// TwinCAT 3 PLC project Testing
// ProgramVersion: 3.1.4026.13
// libraries:
//   Tc2_Standard, * (Beckhoff Automation GmbH)
//   Tc2_System, * (Beckhoff Automation GmbH)
//   Tc3_Component, * (Zerlauth)
//   Tc3_Module, * (Beckhoff Automation GmbH)
//   Tc3_UnitTest, * (Zerlauth)
// project tree:
//   / PlcTask.TcTTO
//   POUs/ MAIN.TcPOU
//   Tests/ FB_ListComponentTests.TcPOU, FB_ListObjectTests.TcPOU, FB_ListStringTests.TcPOU (not stored), FB_MembersTests.TcPOU, FB_ComponentTests.TcPOU (not stored)
// (motion and I/O tree: see PLC project development)
// real-time tasks:
//   TASK PlcTask: cycle T#500ms, priority 21, ADS port 351
//   TASK UnitTestTask: cycle T#1ms, priority 1, ADS port 350
// variable links:

CONFIGURATION Testing
    RESOURCE PLC ON TwinCAT3
        TASK PlcTask(INTERVAL := T#1ms, PRIORITY := 1);
        PROGRAM MAIN WITH PlcTask : MAIN;
    END_RESOURCE
END_CONFIGURATION

// ---- POUs/MAIN.TcPOU
PROGRAM MAIN
VAR
	bInitialise: 			BOOL:= TRUE;
	bExecute: 				BOOL;
	fbTestsuites:			FB_Testsuites;
	fbListObject:			FB_ListObjectTests;
	fbListComponent:		FB_ListComponentTests;
	fbListString:			FB_ListStringTests;
	fbMembers:				FB_MembersTests;
	fbComponentTests:		FB_ComponentTests;
END_VAR

IF bInitialise THEN
	bInitialise:= FALSE;
	fbTestsuites.M_Add(fbListObject.fbTestsuite);
	fbTestsuites.M_Add(fbListComponent.fbTestsuite);
	fbTestsuites.M_Add(fbListString.fbTestsuite);
	fbTestsuites.M_Add(fbMembers.fbTestsuite);
	fbTestsuites.M_Add(fbComponentTests.fbTestsuite);
	fbTestsuites.P_Options.sFilePathName:= 'C:\report.xml';
END_IF

IF bExecute THEN
	bExecute:= fbTestsuites.M_Request(E_Base.Execute);
END_IF

fbTestsuites();


fbListObject();
fbListComponent();
fbListString();
fbMembers();
fbComponentTests();

END_PROGRAM

// ---- Tests/FB_ListObjectTests.TcPOU
FUNCTION_BLOCK FB_ListObjectTests EXTENDS 
VAR_INPUT
END_VAR
VAR_OUTPUT
	fbTestsuite:			FB_Testsuite;
END_VAR
VAR
	fbList:					Tc3_Component.FB_ListObject;
	fbObject:				Tc3_Component.FB_Component;
	iObject:				Tc3_Component.I_Object:= fbObject;
END_VAR

fbTestsuite.P_Property.M_Add('object', 'FB_ListObject');
fbTestsuite.P_Property.M_Add('name', 'Peter Zerlauth');

fbTestsuite();

CASE fbTestsuite.P_Testcase OF
	
	E_Testcase.Start:
		fbTestsuite.P_Assert.M_Equals_DINT(fbList.P_Length, 0, 'P_Length');
		fbTestsuite.M_Testcase('FB_ListObject', T#2S, 'fbList.P_Length', '', 10);	
		
	10:
		fbTestsuite.P_Assert.M_Equals_BOOL(fbList.M_Add(fbObject), TRUE, 'M_Add(fbObject)');
		fbTestsuite.M_Testcase('FB_ListObject', T#2S, 'fbList.M_Add(fbObject)', '', 20);
		
	20:
		fbTestsuite.P_Assert.M_Equals_DINT(fbList.P_Length, 1, 'P_Length');
		fbTestsuite.M_Testcase('FB_ListObject', T#2S, 'fbList.P_Length', '', 30);		
		
	30:
		fbTestsuite.P_Assert.M_Equals_DINT(fbList.M_Find(fbObject), 0, 'M_Find');
		fbTestsuite.M_Testcase('FB_ListObject', T#2S, 'fbList.M_Find(fbObject)', '', 40);
		
	40:

		fbTestsuite.P_Assert.M_Equals_BOOL(TRUE, __QUERYINTERFACE(fbList.M_Index(0), iObject), 'M_Index');
		fbTestsuite.M_Testcase('FB_ListObject', T#2S, 'fbList.M_Index(1)', '', 50);
		
	50:
		fbTestsuite.P_Assert.M_Equals_BOOL(fbList.M_Remove(fbObject), TRUE, 'M_Remove');
		fbTestsuite.M_Testcase('FB_ListObject', T#2S, 'fbList.M_Remove(fbObject', '', 60);		

	60:
		fbTestsuite.P_Assert.M_Equals_DINT(fbList.P_Length, 0, 'P_Length');
		fbTestsuite.M_Testcase('FB_ListObject', T#2S, 'fbList.P_Length', '', 70);
		
	70:
		fbTestsuite.P_Assert.M_Equals_BOOL(fbList.M_Add(fbObject), TRUE, 'M_Add(fbObject)');
		fbTestsuite.M_Testcase('FB_ListObject', T#2S, 'fbList.M_Add(fbObject)', '', 80);

	80:
		fbTestsuite.P_Assert.M_Equals_DINT(fbList.P_Length, 1, 'P_Length');
		fbTestsuite.M_Testcase('FB_ListObject', T#2S, 'fbList.P_Length', '', 90);
		
	90:
		fbTestsuite.P_Assert.M_Equals_BOOL(fbList.M_Clear(), TRUE, 'M_Clear()');
		fbTestsuite.M_Testcase('FB_ListObject', T#2S, 'fbList.M_Clear()', '', 100);		
	
	100:
		fbTestsuite.P_Assert.M_Equals_DINT(fbList.P_Length, 0, 'P_Length');
		fbTestsuite.M_Testcase('FB_ListObject', T#2S, 'fbList.P_Length', '', E_Testcase.Done);
		
	E_Testcase.Done:
		;
END_CASE

END_FUNCTION_BLOCK

// ---- Tests/FB_ListComponentTests.TcPOU
FUNCTION_BLOCK FB_ListComponentTests EXTENDS 
VAR_INPUT
END_VAR
VAR_OUTPUT
	fbTestsuite:			FB_Testsuite;
END_VAR
VAR
	fbList:					Tc3_Component.FB_ListComponent;
	fbObject:				Tc3_Component.FB_Component;
	iObject:				Tc3_Component.I_Element:= fbObject;
END_VAR

fbTestsuite.P_Property.M_Add('object', 'FB_ListComponent');
fbTestsuite.P_Property.M_Add('name', 'Peter Zerlauth');

fbTestsuite();

CASE fbTestsuite.P_Testcase OF
	
	E_Testcase.Start:
		fbTestsuite.P_Assert.M_Equals_DINT(fbList.P_Length, 0, 'P_Length');
		fbTestsuite.M_Testcase('FB_ListComponent', T#2S, 'fbList.P_Length', '', 10);	
		
	10:
		fbTestsuite.P_Assert.M_Equals_BOOL(fbList.M_Add(fbObject), TRUE, 'M_Add(fbObject)');
		fbTestsuite.M_Testcase('FB_ListComponent', T#2S, 'fbList.M_Add(fbObject)', '', 20);
		
	20:
		fbTestsuite.P_Assert.M_Equals_DINT(fbList.P_Length, 1, 'P_Length');
		fbTestsuite.M_Testcase('FB_ListComponent', T#2S, 'fbList.P_Length', '', 30);		
		
	30:
		fbTestsuite.P_Assert.M_Equals_DINT(fbList.M_Find(fbObject), 0, 'M_Find');
		fbTestsuite.M_Testcase('FB_ListComponent', T#2S, 'fbList.M_Find(fbObject)', '', 40);
		
	40:

		fbTestsuite.P_Assert.M_Equals_BOOL(TRUE, __QUERYINTERFACE(fbList.M_Index(0), iObject), 'M_Index');
		fbTestsuite.M_Testcase('FB_ListComponent', T#2S, 'fbList.M_Index(1)', '', 50);
		
	50:
		fbTestsuite.P_Assert.M_Equals_BOOL(fbList.M_Remove(fbObject), TRUE, 'M_Remove');
		fbTestsuite.M_Testcase('FB_ListComponent', T#2S, 'fbList.M_Remove(fbObject', '', 60);		

	60:
		fbTestsuite.P_Assert.M_Equals_DINT(fbList.P_Length, 0, 'P_Length');
		fbTestsuite.M_Testcase('FB_ListComponent', T#2S, 'fbList.P_Length', '', 70);
		
	70:
		fbTestsuite.P_Assert.M_Equals_BOOL(fbList.M_Add(fbObject), TRUE, 'M_Add(fbObject)');
		fbTestsuite.M_Testcase('FB_ListComponent', T#2S, 'fbList.M_Add(fbObject)', '', 80);

	80:
		fbTestsuite.P_Assert.M_Equals_DINT(fbList.P_Length, 1, 'P_Length');
		fbTestsuite.M_Testcase('FB_ListComponent', T#2S, 'fbList.P_Length', '', 90);
		
	90:
		fbTestsuite.P_Assert.M_Equals_BOOL(fbList.M_Clear(), TRUE, 'M_Clear()');
		fbTestsuite.M_Testcase('FB_ListComponent', T#2S, 'fbList.M_Clear()', '', 100);		
	
	100:
		fbTestsuite.P_Assert.M_Equals_DINT(fbList.P_Length, 0, 'P_Length');
		fbTestsuite.M_Testcase('FB_ListComponent', T#2S, 'fbList.P_Length', '', E_Testcase.Done);
		
	E_Testcase.Done:
		;
END_CASE

END_FUNCTION_BLOCK

// ---- Tests/FB_MembersTests.TcPOU
FUNCTION_BLOCK FB_MembersTests EXTENDS 
VAR_INPUT
END_VAR
VAR_OUTPUT
	fbTestsuite:			FB_Testsuite;
END_VAR
VAR
	fbList:					Tc3_Component.FB_Members;
	fbObject1:				Tc3_Component.FB_Component;
	fbObject2:				Tc3_Component.FB_Component;
END_VAR

fbTestsuite.P_Property.M_Add('object', 'FB_Members');
fbTestsuite.P_Property.M_Add('name', 'Peter Zerlauth');

fbTestsuite();

fbObject1();
fbObject2();

CASE fbTestsuite.P_Testcase OF
	
	E_Testcase.Start:
		fbList.M_Clear();
		fbTestsuite.P_Assert.M_Equals_DINT(fbList.P_Length, 0, 'P_Length');
		fbTestsuite.M_Testcase('FB_Members', T#2S, 'fbList.P_Length', '', 10);	
		
	10:
		fbTestsuite.P_Assert.M_Equals_BOOL(fbList.M_Add(fbObject1), TRUE, 'M_Add(fbObject1)');
		fbTestsuite.P_Assert.M_Equals_BOOL(fbList.M_Add(fbObject2), TRUE, 'M_Add(fbObject2)');
		fbTestsuite.P_Assert.M_Equals_DINT(fbList.P_Length, 2, 'P_Length');
		fbTestsuite.M_Testcase('FB_Members', T#2S, 'fbList.M_Add(fbObject)', '', 20);
		
	20:
		fbTestsuite.P_Assert.M_Equals_BOOL(fbList.M_Start(), 1, 'M_Start()');
		fbTestsuite.P_Assert.M_Equals_DINT(fbObject1.P_State, E_State.Execute, 'P_State');
		fbTestsuite.M_Testcase('FB_Members', T#2S, 'fbList.M_Start()', '', 30);		
		
	30:
		fbTestsuite.P_Assert.M_Equals_BOOL(fbList.M_Error(), 1, 'M_Error()');
		fbTestsuite.P_Assert.M_Equals_DINT(fbObject1.P_State, E_State.Stopped, 'P_State');
		fbTestsuite.M_Testcase('FB_Members', T#2S, 'fbList.M_Error()', '', 40);
		
	40:

		fbTestsuite.P_Assert.M_Equals_BOOL(fbList.M_Reset(), 1, 'M_Reset()');
		fbTestsuite.P_Assert.M_Equals_DINT(fbObject1.P_State, E_State.Idle, 'P_State');
		fbTestsuite.M_Testcase('FB_Members', T#2S, 'fbList.M_Reset()', '', 50);
		
	50:
		fbTestsuite.P_Assert.M_Equals_BOOL(fbList.M_Start(), 1, 'M_Start()');
		fbTestsuite.P_Assert.M_Equals_DINT(fbObject1.P_State, E_State.Execute, 'P_State');
		fbTestsuite.M_Testcase('FB_Members', T#2S, 'fbList.M_Start()', '', 60);		

	60:
		fbTestsuite.P_Assert.M_Equals_BOOL(fbList.M_Abort(), 1, 'M_Abort()');
		fbTestsuite.P_Assert.M_Equals_DINT(fbObject1.P_State, E_State.Aborted, 'P_State');
		fbTestsuite.M_Testcase('FB_Members', T#2S, 'fbList.M_Abort()', '', 70);
		
	70:
		fbTestsuite.P_Assert.M_Equals_BOOL(fbList.M_Reset(), 1, 'M_Reset()');
		fbTestsuite.P_Assert.M_Equals_DINT(fbObject1.P_State, E_State.Idle, 'P_State');
		fbTestsuite.M_Testcase('FB_Members', T#2S, 'fbList.M_Reset()', '',E_Testcase.Done);
		
	E_Testcase.Done:
		;
END_CASE

END_FUNCTION_BLOCK
